TYPE "Prod_Part_Done"
VERSION : 0.1
// Block: Prod_Part_Done
   STRUCT
      Done : Bool;
      LeadCut : Bool;
      Weld : Bool;
      Tick_Mark : Bool;
      Trace_Mark : Bool;
      P_ID : DInt;
      O_ID : DInt;
      Part_LenMeas : Real;
   END_STRUCT;

END_TYPE
